(* Logix 5000 project; controller Receptivo vendor 1 type 14 code 106 rev 30.11; software revision 30.00; part 7 of 10 *)
(* tags used below, declared in another part *)
   Final_Print_1 : BOOL;
   Final_Print_2 : BOOL;
   Final_Print_3 : BOOL;
   Final_Print_4 : BOOL;
   ons_imprimiendo : BOOL;
   ons_nuevo_dia : BOOL;
   ons_print1 : BOOL;
   ons_print1_aux : BOOL;
   ons_print2 : BOOL;
   ons_print2_2 : BOOL;
   ons_print3 : BOOL;
   ons_print3_aux : BOOL;
   ons_print4 : BOOL;
   ons_print4_aux : BOOL;
   Print1_Ejecute : BOOL;
   Print1_OK : BOOL;
   Print2_Ejecute : BOOL;
   Print2_OK : BOOL;
   Print3_Ejecute : BOOL;
   Print3_OK : BOOL;
   Print4_Ejecute : BOOL;
   Print4_OK : BOOL;
   Printing_1 : BOOL;
   Printing_2 : BOOL;
   Printing_3 : BOOL;
   Printing_4 : BOOL;
   Salida_Cola_Est_1 : UDT_COLA;
   Salida_Cola_Est_2 : UDT_COLA;
   Salida_Cola_Est_3 : UDT_COLA;
   Salida_Cola_Est_4 : UDT_COLA;
   Actualiza1_Timer : TIMER;
   Actualiza2_Timer : TIMER;
   Actualiza3_Timer : TIMER;
   Actualiza4_Timer : TIMER;
   Actualiza_Reporte_1 : BOOL;
   Actualiza_Reporte_2 : BOOL;
   Actualiza_Reporte_3 : BOOL;
   Actualiza_Reporte_4 : BOOL;
   Ano_Biciesto : INT;
   Bit_Medianoche : BOOL;
   Cajas_Calculadas_Estacion_1 : REAL;
   Cajas_Calculadas_Estacion_2 : REAL;
   Cajas_Calculadas_Estacion_3 : REAL;
   Cajas_Calculadas_Estacion_4 : REAL;
   Cajas_CalculadasG_Estacion_1 : REAL;
   Cajas_CalculadasG_Estacion_2 : REAL;
   Cajas_CalculadasG_Estacion_3 : REAL;
   Cajas_CalculadasG_Estacion_4 : REAL;
   Calendario : Hora_y_Fecha;
   Cantidad_de_Productos : DINT;
   CINCO : SINT;
   Clima_1 : DINT;
   Cola_Estacion_1 : UDT_COLA[100];
   Cola_Estacion_1_A : UDT_COLA[100];
   Cola_Estacion_2 : UDT_COLA[100];
   Cola_Estacion_2_A : UDT_COLA[100];
   Cola_Estacion_3 : UDT_COLA[100];
   Cola_Estacion_3_A : UDT_COLA[100];
   Cola_Estacion_4 : UDT_COLA[100];
   Cola_Estacion_4_A : UDT_COLA[100];
   Consecutivo : INT;
   Contador_Consecutivo : COUNTER;
   Control_Cola_Est1 : CONTROL;
   Control_Cola_Est2 : CONTROL;
   Control_Cola_Est3 : CONTROL;
   Control_Cola_Est4 : CONTROL;
   Counter_R_Estacion1 : COUNTER;
   Counter_R_Estacion2 : COUNTER;
   Counter_R_Estacion3 : COUNTER;
   Counter_R_Estacion4 : COUNTER;
   CUATRO : SINT;
   Dia_del_Ano : INT;
   DOS : SINT;
   Espacios : STRING;
   Estacion_1_GCola : UDT_COLA;
   Estacion_1_GCola_1 : UDT_COLA;
   Estacion_1_General : UDT_GENERAL;
   Estacion_1_Resumen : UDT_COLA[20];
   Estacion_1_Resumen_A : UDT_COLA[20];
   Estacion_2_GCola : UDT_COLA;
   Estacion_2_GCola_1 : UDT_COLA;
   Estacion_2_General : UDT_GENERAL;
   Estacion_2_Resumen : UDT_COLA[20];
   Estacion_2_Resumen_A : UDT_COLA[20];
   Estacion_3_GCola : UDT_COLA;
   Estacion_3_GCola_1 : UDT_COLA;
   Estacion_3_General : UDT_GENERAL;
   Estacion_3_Resumen : UDT_COLA[20];
   Estacion_3_Resumen_A : UDT_COLA[20];
   Estacion_4_GCola : UDT_COLA;
   Estacion_4_GCola_1 : UDT_COLA;
   Estacion_4_General : UDT_GENERAL;
   Estacion_4_Resumen : UDT_COLA[20];
   Estacion_4_Resumen_A : UDT_COLA[20];
   Hoy : DINT;
   Impreso_1 : BOOL;
   Impreso_2 : BOOL;
   Impreso_3 : BOOL;
   Impreso_4 : BOOL;
   Imprimiendo_1 : BOOL;
   Imprimiendo_1_Timer : TIMER;
   Imprimiendo_2 : BOOL;
   Imprimiendo_2_Timer : TIMER;
   Imprimiendo_3 : BOOL;
   Imprimiendo_3_Timer : TIMER;
   Imprimiendo_4 : BOOL;
   Imprimiendo_4_Timer : TIMER;
   Index_Productos : DINT;
   Listado : INT;
   Listado_A : INT;
   Lote : DINT;
   Mes_dias : INT[13];
   new_day : BOOL;
   Num_Cajas_Reales_1 : DINT;
   Num_Cajas_Reales_2 : DINT;
   Num_Cajas_Reales_3 : DINT;
   Num_Cajas_Reales_4 : DINT;
   ons_add : BOOL;
   ons_add2 : BOOL;
   ons_add3 : BOOL;
   ons_add4 : BOOL;
   Ons_Corte_Dia : BOOL;
   Ons_NP : BOOL;
   Ons_NP2 : BOOL;
   Ons_NP3 : BOOL;
   Ons_NP4 : BOOL;
   ONS_Reporte_Dia : BOOL;
   Operador_1 : DINT;
   Peso_OK_Estacion_1 : BOOL;
   Peso_OK_Estacion_2 : BOOL;
   Peso_OK_Estacion_3 : BOOL;
   Peso_OK_Estacion_4 : BOOL;
   PESO_REAL_1 : DINT;
   PESO_REAL_2 : DINT;
   PESO_REAL_3 : DINT;
   PESO_REAL_4 : DINT;
   Print_1 : BOOL;
   Print_2 : BOOL;
   Print_3 : BOOL;
   Print_4 : BOOL;
   Printing_Enable : BOOL;
   Producto1 : UDT_Inventario;
   Producto2 : UDT_Inventario;
   Producto3 : UDT_Inventario;
   Producto4 : UDT_Inventario;
   Productos : UDT_Maestro[300];
   Prueba : UDT_COLA[3];
   Prueba_Bit : BOOL;
   Prueba_Index : DINT;
   Prueba_X : BOOL;
   QAD_Auxiliar_Est1 : STRING;
   QAD_Auxiliar_Est2 : STRING;
   QAD_Auxiliar_Est3 : STRING;
   QAD_Auxiliar_Est4 : STRING;
   Report_Con1 : BOOL;
   Reporte_Dia_Lach : BOOL;
   Reporte_Dia_Timer : TIMER;
   time_new : TIMER;
   TRES : SINT;
   try : BOOL;
   UNO : SINT;
   Zero : DINT;
(* MainProgram, continued *)

ROUTINE Impresion_1   (* ladder *)
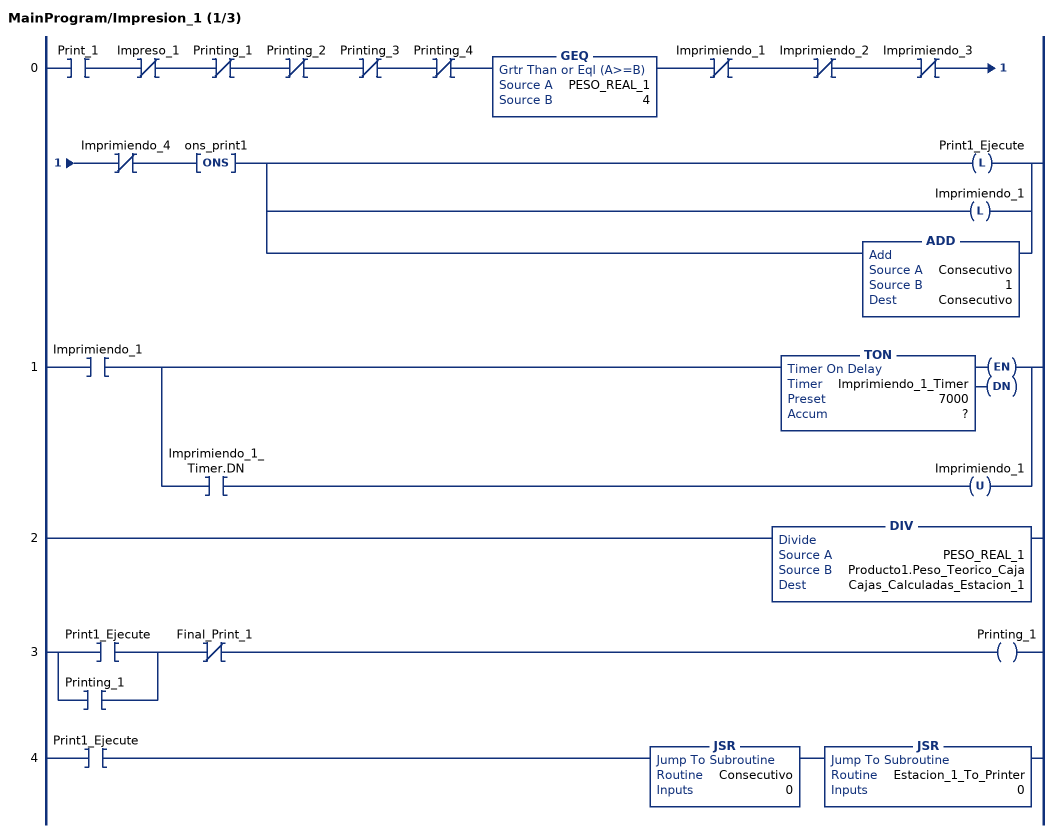
   0: XIC(Print_1)XIO(Impreso_1)XIO(Printing_1)XIO(Printing_2)XIO(Printing_3)XIO(Printing_4)GEQ(PESO_REAL_1,4)XIO(Imprimiendo_1)XIO(Imprimiendo_2)XIO(Imprimiendo_3)XIO(Imprimiendo_4)ONS(ons_print1)[OTL(Print1_Ejecute) ,OTL(Imprimiendo_1) ,ADD(Consecutivo,1,Consecutivo) ];
   1: XIC(Imprimiendo_1)[TON(Imprimiendo_1_Timer,?,?) ,XIC(Imprimiendo_1_Timer.DN) OTU(Imprimiendo_1) ];
   2: DIV(PESO_REAL_1,Producto1.Peso_Teorico_Caja,Cajas_Calculadas_Estacion_1);
   3: [XIC(Print1_Ejecute) ,XIC(Printing_1) ]XIO(Final_Print_1)OTE(Printing_1);
   4: XIC(Print1_Ejecute)JSR(Consecutivo,0)JSR(Estacion_1_To_Printer,0);
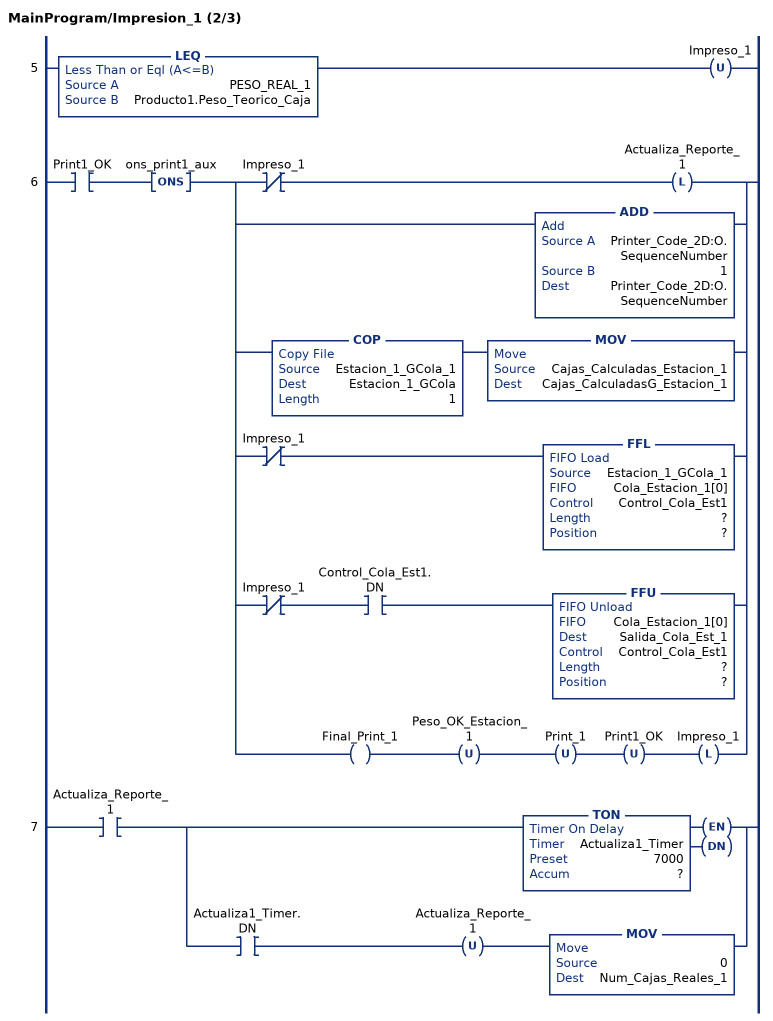
   5: LEQ(PESO_REAL_1,Producto1.Peso_Teorico_Caja)OTU(Impreso_1);
   6: XIC(Print1_OK)ONS(ons_print1_aux)[XIO(Impreso_1) OTL(Actualiza_Reporte_1) ,ADD(Printer_Code_2D:O.SequenceNumber,1,Printer_Code_2D:O.SequenceNumber) ,COP(Estacion_1_GCola_1,Estacion_1_GCola,1) MOV(Cajas_Calculadas_Estacion_1,Cajas_CalculadasG_Estacion_1) ,XIO(Impreso_1) FFL(Estacion_1_GCola_1,Cola_Estacion_1[0],Control_Cola_Est1,?,?) ,XIO(Impreso_1) XIC(Control_Cola_Est1.DN) FFU(Cola_Estacion_1[0],Salida_Cola_Est_1,Control_Cola_Est1,?,?) ,OTE(Final_Print_1) OTU(Peso_OK_Estacion_1) OTU(Print_1) OTU(Print1_OK) OTL(Impreso_1) ];
   7: XIC(Actualiza_Reporte_1)[TON(Actualiza1_Timer,?,?) ,XIC(Actualiza1_Timer.DN) OTU(Actualiza_Reporte_1) MOV(0,Num_Cajas_Reales_1) ];
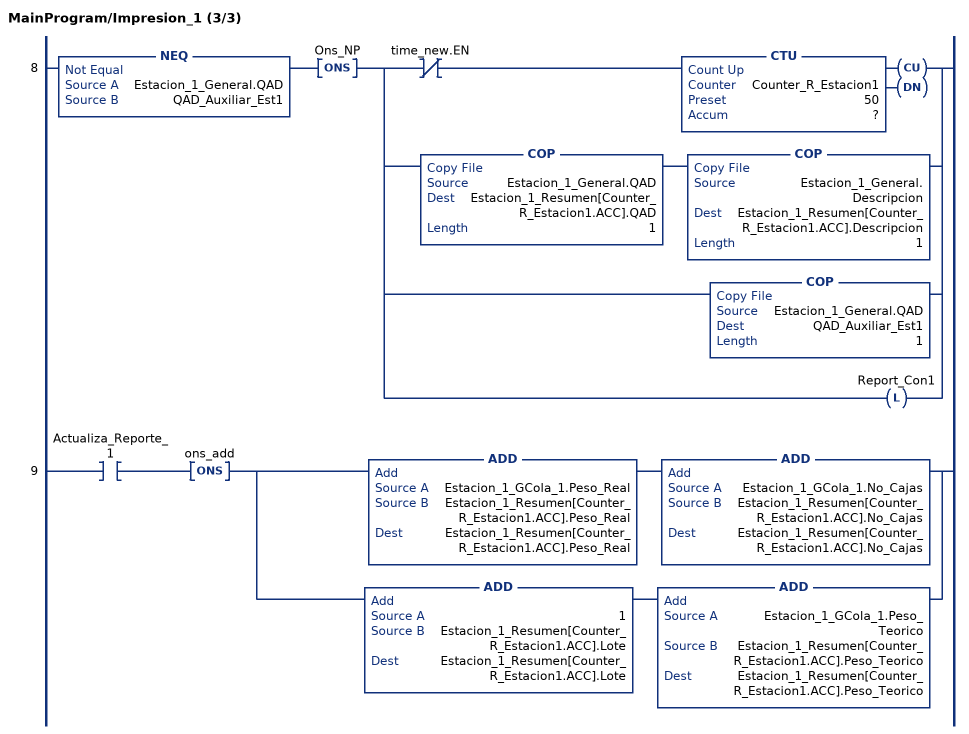
   8: NEQ(Estacion_1_General.QAD,QAD_Auxiliar_Est1)ONS(Ons_NP)[XIO(time_new.EN) CTU(Counter_R_Estacion1,?,?) ,COP(Estacion_1_General.QAD,Estacion_1_Resumen[Counter_R_Estacion1.ACC].QAD,1) COP(Estacion_1_General.Descripcion,Estacion_1_Resumen[Counter_R_Estacion1.ACC].Descripcion,1) ,COP(Estacion_1_General.QAD,QAD_Auxiliar_Est1,1) ,OTL(Report_Con1) ];
   9: XIC(Actualiza_Reporte_1)ONS(ons_add)[ADD(Estacion_1_GCola_1.Peso_Real,Estacion_1_Resumen[Counter_R_Estacion1.ACC].Peso_Real,Estacion_1_Resumen[Counter_R_Estacion1.ACC].Peso_Real) ADD(Estacion_1_GCola_1.No_Cajas,Estacion_1_Resumen[Counter_R_Estacion1.ACC].No_Cajas,Estacion_1_Resumen[Counter_R_Estacion1.ACC].No_Cajas) ,ADD(1,Estacion_1_Resumen[Counter_R_Estacion1.ACC].Lote,Estacion_1_Resumen[Counter_R_Estacion1.ACC].Lote) ADD(Estacion_1_GCola_1.Peso_Teorico,Estacion_1_Resumen[Counter_R_Estacion1.ACC].Peso_Teorico,Estacion_1_Resumen[Counter_R_Estacion1.ACC].Peso_Teorico) ];
END_ROUTINE

ROUTINE Impresion_2   (* ladder *)
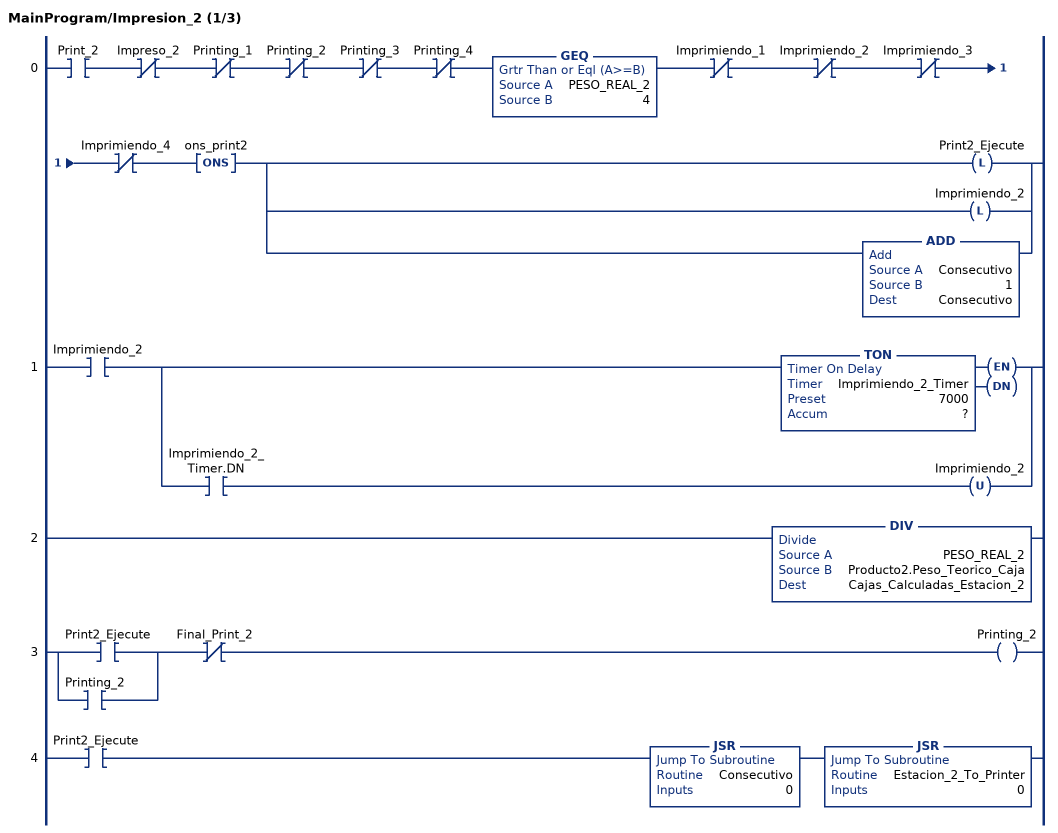
   0: XIC(Print_2)XIO(Impreso_2)XIO(Printing_1)XIO(Printing_2)XIO(Printing_3)XIO(Printing_4)GEQ(PESO_REAL_2,4)XIO(Imprimiendo_1)XIO(Imprimiendo_2)XIO(Imprimiendo_3)XIO(Imprimiendo_4)ONS(ons_print2)[OTL(Print2_Ejecute) ,OTL(Imprimiendo_2) ,ADD(Consecutivo,1,Consecutivo) ];
   1: XIC(Imprimiendo_2)[TON(Imprimiendo_2_Timer,?,?) ,XIC(Imprimiendo_2_Timer.DN) OTU(Imprimiendo_2) ];
   2: DIV(PESO_REAL_2,Producto2.Peso_Teorico_Caja,Cajas_Calculadas_Estacion_2);
   3: [XIC(Print2_Ejecute) ,XIC(Printing_2) ]XIO(Final_Print_2)OTE(Printing_2);
   4: XIC(Print2_Ejecute)JSR(Consecutivo,0)JSR(Estacion_2_To_Printer,0);
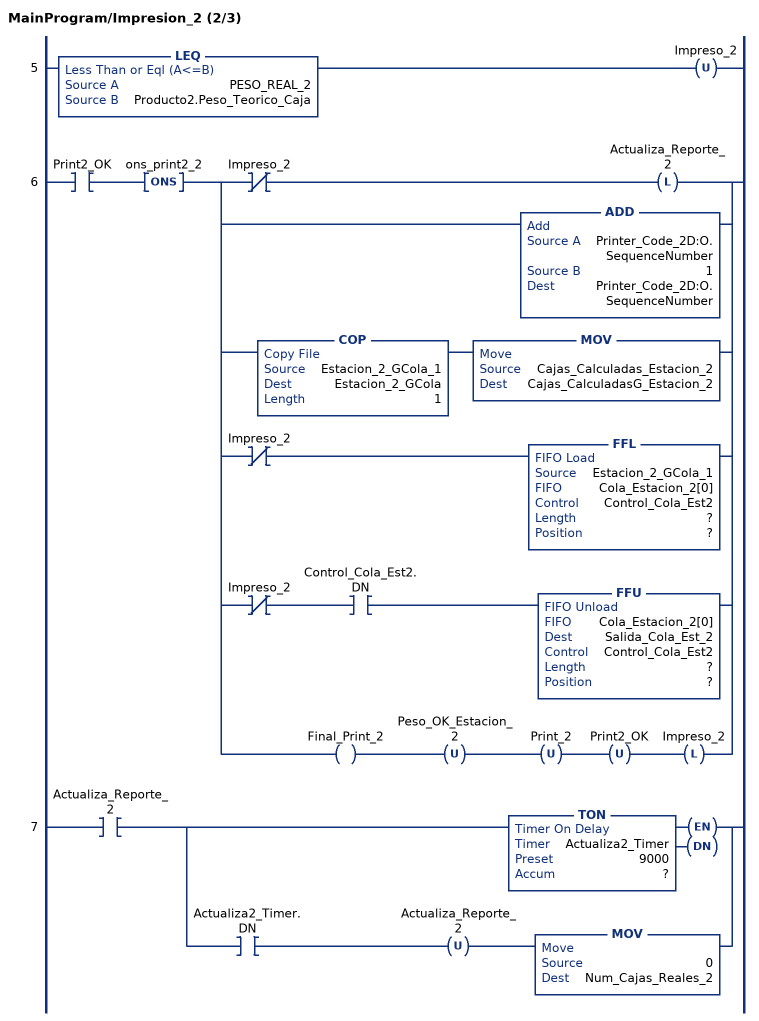
   5: LEQ(PESO_REAL_2,Producto2.Peso_Teorico_Caja)OTU(Impreso_2);
   6: XIC(Print2_OK)ONS(ons_print2_2)[XIO(Impreso_2) OTL(Actualiza_Reporte_2) ,ADD(Printer_Code_2D:O.SequenceNumber,1,Printer_Code_2D:O.SequenceNumber) ,COP(Estacion_2_GCola_1,Estacion_2_GCola,1) MOV(Cajas_Calculadas_Estacion_2,Cajas_CalculadasG_Estacion_2) ,XIO(Impreso_2) FFL(Estacion_2_GCola_1,Cola_Estacion_2[0],Control_Cola_Est2,?,?) ,XIO(Impreso_2) XIC(Control_Cola_Est2.DN) FFU(Cola_Estacion_2[0],Salida_Cola_Est_2,Control_Cola_Est2,?,?) ,OTE(Final_Print_2) OTU(Peso_OK_Estacion_2) OTU(Print_2) OTU(Print2_OK) OTL(Impreso_2) ];
   7: XIC(Actualiza_Reporte_2)[TON(Actualiza2_Timer,?,?) ,XIC(Actualiza2_Timer.DN) OTU(Actualiza_Reporte_2) MOV(0,Num_Cajas_Reales_2) ];
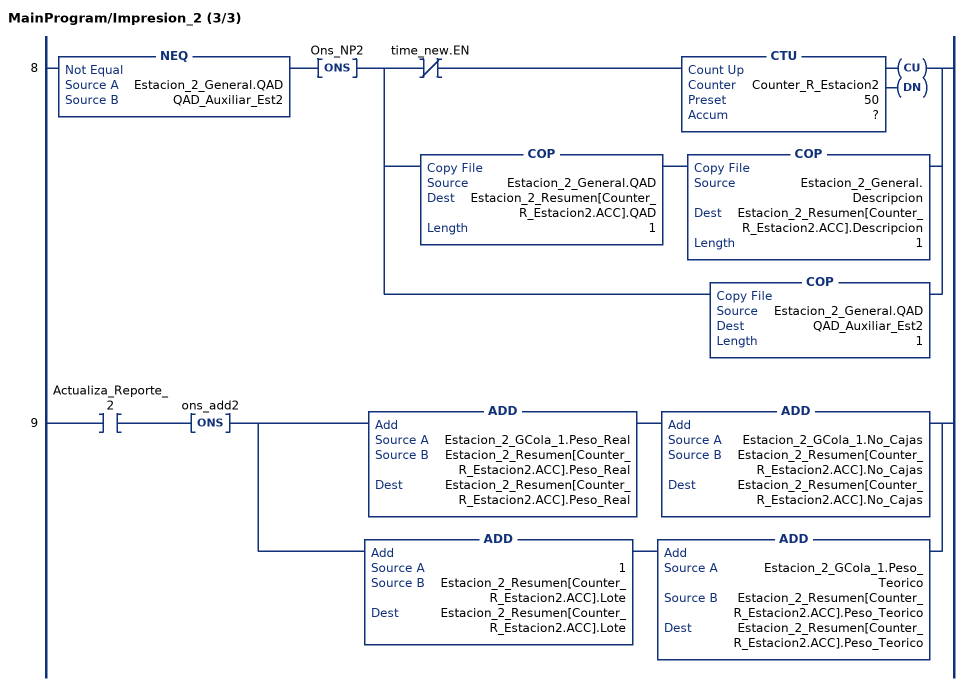
   8: NEQ(Estacion_2_General.QAD,QAD_Auxiliar_Est2)ONS(Ons_NP2)[XIO(time_new.EN) CTU(Counter_R_Estacion2,?,?) ,COP(Estacion_2_General.QAD,Estacion_2_Resumen[Counter_R_Estacion2.ACC].QAD,1) COP(Estacion_2_General.Descripcion,Estacion_2_Resumen[Counter_R_Estacion2.ACC].Descripcion,1) ,COP(Estacion_2_General.QAD,QAD_Auxiliar_Est2,1) ];
   9: XIC(Actualiza_Reporte_2)ONS(ons_add2)[ADD(Estacion_2_GCola_1.Peso_Real,Estacion_2_Resumen[Counter_R_Estacion2.ACC].Peso_Real,Estacion_2_Resumen[Counter_R_Estacion2.ACC].Peso_Real) ADD(Estacion_2_GCola_1.No_Cajas,Estacion_2_Resumen[Counter_R_Estacion2.ACC].No_Cajas,Estacion_2_Resumen[Counter_R_Estacion2.ACC].No_Cajas) ,ADD(1,Estacion_2_Resumen[Counter_R_Estacion2.ACC].Lote,Estacion_2_Resumen[Counter_R_Estacion2.ACC].Lote) ADD(Estacion_2_GCola_1.Peso_Teorico,Estacion_2_Resumen[Counter_R_Estacion2.ACC].Peso_Teorico,Estacion_2_Resumen[Counter_R_Estacion2.ACC].Peso_Teorico) ];
END_ROUTINE

ROUTINE Impresion_3   (* ladder *)
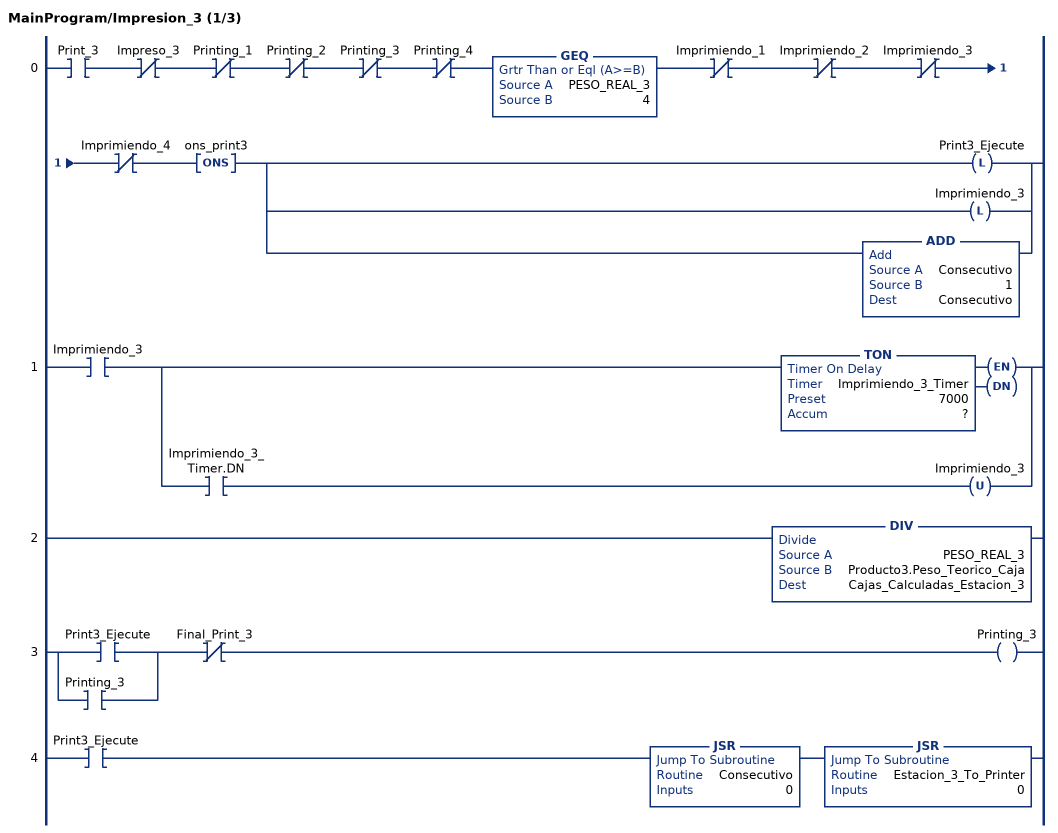
   0: XIC(Print_3)XIO(Impreso_3)XIO(Printing_1)XIO(Printing_2)XIO(Printing_3)XIO(Printing_4)GEQ(PESO_REAL_3,4)XIO(Imprimiendo_1)XIO(Imprimiendo_2)XIO(Imprimiendo_3)XIO(Imprimiendo_4)ONS(ons_print3)[OTL(Print3_Ejecute) ,OTL(Imprimiendo_3) ,ADD(Consecutivo,1,Consecutivo) ];
   1: XIC(Imprimiendo_3)[TON(Imprimiendo_3_Timer,?,?) ,XIC(Imprimiendo_3_Timer.DN) OTU(Imprimiendo_3) ];
   2: DIV(PESO_REAL_3,Producto3.Peso_Teorico_Caja,Cajas_Calculadas_Estacion_3);
   3: [XIC(Print3_Ejecute) ,XIC(Printing_3) ]XIO(Final_Print_3)OTE(Printing_3);
   4: XIC(Print3_Ejecute)JSR(Consecutivo,0)JSR(Estacion_3_To_Printer,0);
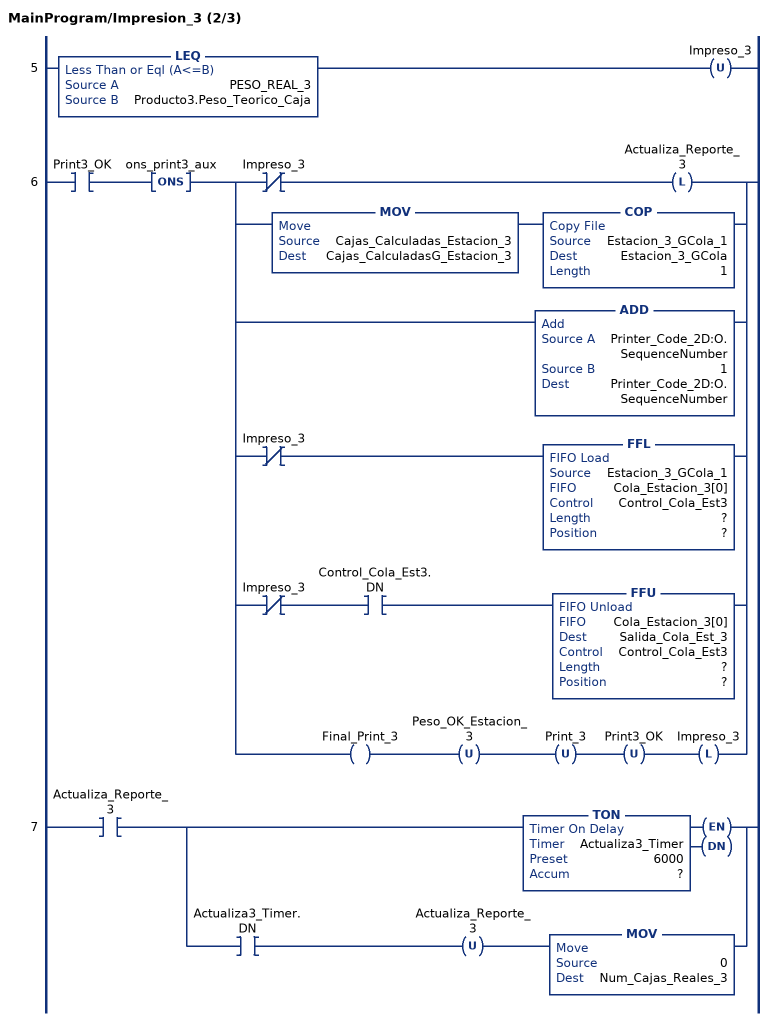
   5: LEQ(PESO_REAL_3,Producto3.Peso_Teorico_Caja)OTU(Impreso_3);
   6: XIC(Print3_OK)ONS(ons_print3_aux)[XIO(Impreso_3) OTL(Actualiza_Reporte_3) ,MOV(Cajas_Calculadas_Estacion_3,Cajas_CalculadasG_Estacion_3) COP(Estacion_3_GCola_1,Estacion_3_GCola,1) ,ADD(Printer_Code_2D:O.SequenceNumber,1,Printer_Code_2D:O.SequenceNumber) ,XIO(Impreso_3) FFL(Estacion_3_GCola_1,Cola_Estacion_3[0],Control_Cola_Est3,?,?) ,XIO(Impreso_3) XIC(Control_Cola_Est3.DN) FFU(Cola_Estacion_3[0],Salida_Cola_Est_3,Control_Cola_Est3,?,?) ,OTE(Final_Print_3) OTU(Peso_OK_Estacion_3) OTU(Print_3) OTU(Print3_OK) OTL(Impreso_3) ];
   7: XIC(Actualiza_Reporte_3)[TON(Actualiza3_Timer,?,?) ,XIC(Actualiza3_Timer.DN) OTU(Actualiza_Reporte_3) MOV(0,Num_Cajas_Reales_3) ];
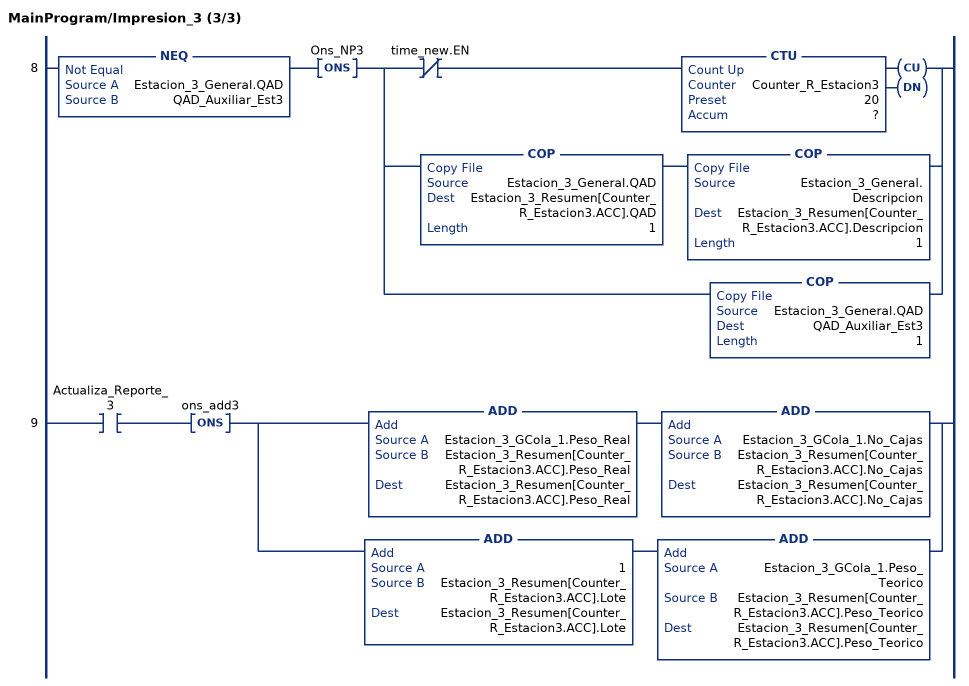
   8: NEQ(Estacion_3_General.QAD,QAD_Auxiliar_Est3)ONS(Ons_NP3)[XIO(time_new.EN) CTU(Counter_R_Estacion3,?,?) ,COP(Estacion_3_General.QAD,Estacion_3_Resumen[Counter_R_Estacion3.ACC].QAD,1) COP(Estacion_3_General.Descripcion,Estacion_3_Resumen[Counter_R_Estacion3.ACC].Descripcion,1) ,COP(Estacion_3_General.QAD,QAD_Auxiliar_Est3,1) ];
   9: XIC(Actualiza_Reporte_3)ONS(ons_add3)[ADD(Estacion_3_GCola_1.Peso_Real,Estacion_3_Resumen[Counter_R_Estacion3.ACC].Peso_Real,Estacion_3_Resumen[Counter_R_Estacion3.ACC].Peso_Real) ADD(Estacion_3_GCola_1.No_Cajas,Estacion_3_Resumen[Counter_R_Estacion3.ACC].No_Cajas,Estacion_3_Resumen[Counter_R_Estacion3.ACC].No_Cajas) ,ADD(1,Estacion_3_Resumen[Counter_R_Estacion3.ACC].Lote,Estacion_3_Resumen[Counter_R_Estacion3.ACC].Lote) ADD(Estacion_3_GCola_1.Peso_Teorico,Estacion_3_Resumen[Counter_R_Estacion3.ACC].Peso_Teorico,Estacion_3_Resumen[Counter_R_Estacion3.ACC].Peso_Teorico) ];
END_ROUTINE

ROUTINE Impresion_4   (* ladder *)
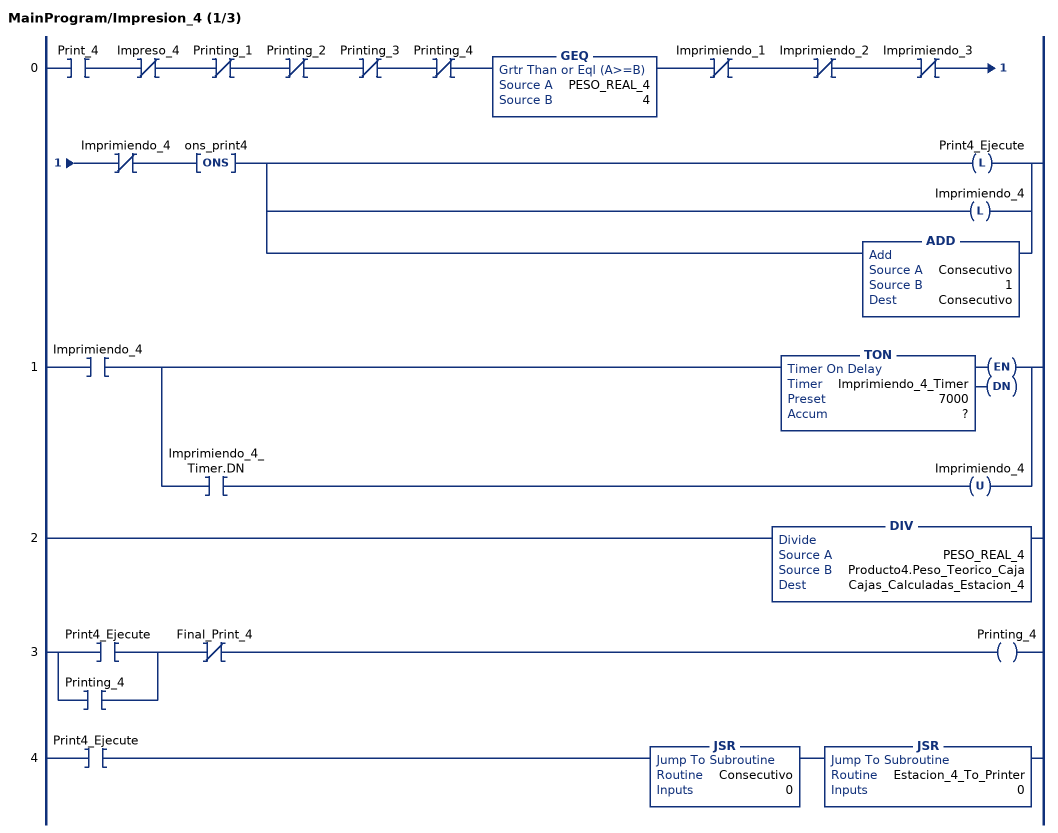
   0: XIC(Print_4)XIO(Impreso_4)XIO(Printing_1)XIO(Printing_2)XIO(Printing_3)XIO(Printing_4)GEQ(PESO_REAL_4,4)XIO(Imprimiendo_1)XIO(Imprimiendo_2)XIO(Imprimiendo_3)XIO(Imprimiendo_4)ONS(ons_print4)[OTL(Print4_Ejecute) ,OTL(Imprimiendo_4) ,ADD(Consecutivo,1,Consecutivo) ];
   1: XIC(Imprimiendo_4)[TON(Imprimiendo_4_Timer,?,?) ,XIC(Imprimiendo_4_Timer.DN) OTU(Imprimiendo_4) ];
   2: DIV(PESO_REAL_4,Producto4.Peso_Teorico_Caja,Cajas_Calculadas_Estacion_4);
   3: [XIC(Print4_Ejecute) ,XIC(Printing_4) ]XIO(Final_Print_4)OTE(Printing_4);
   4: XIC(Print4_Ejecute)JSR(Consecutivo,0)JSR(Estacion_4_To_Printer,0);
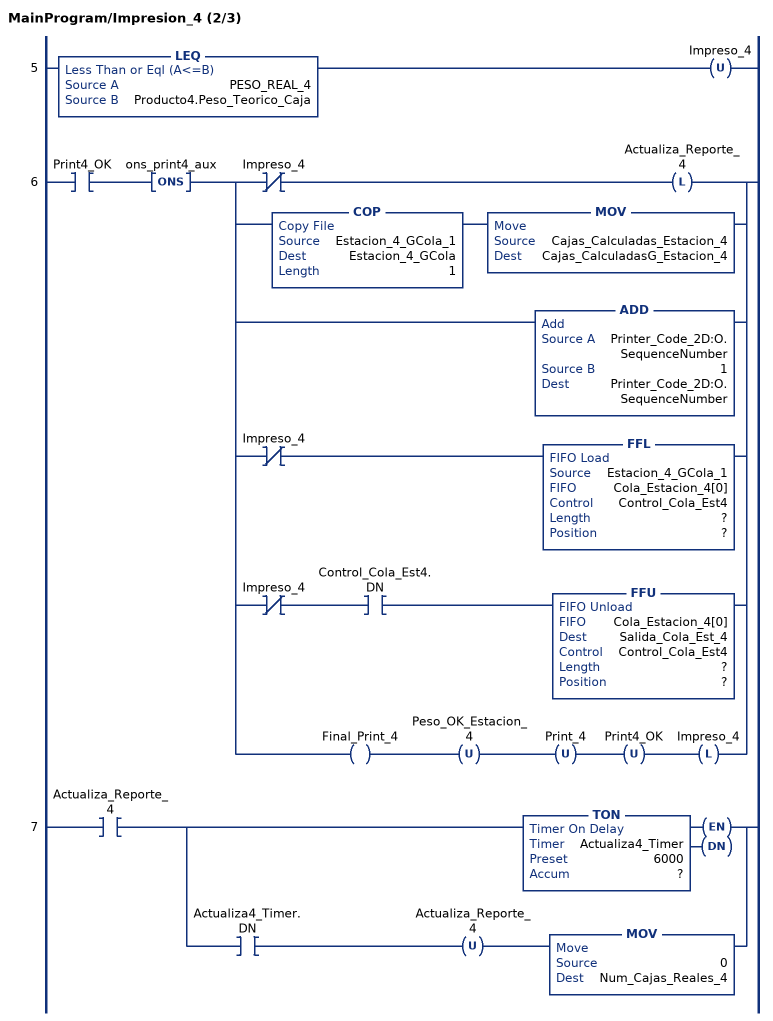
   5: LEQ(PESO_REAL_4,Producto4.Peso_Teorico_Caja)OTU(Impreso_4);
   6: XIC(Print4_OK)ONS(ons_print4_aux)[XIO(Impreso_4) OTL(Actualiza_Reporte_4) ,COP(Estacion_4_GCola_1,Estacion_4_GCola,1) MOV(Cajas_Calculadas_Estacion_4,Cajas_CalculadasG_Estacion_4) ,ADD(Printer_Code_2D:O.SequenceNumber,1,Printer_Code_2D:O.SequenceNumber) ,XIO(Impreso_4) FFL(Estacion_4_GCola_1,Cola_Estacion_4[0],Control_Cola_Est4,?,?) ,XIO(Impreso_4) XIC(Control_Cola_Est4.DN) FFU(Cola_Estacion_4[0],Salida_Cola_Est_4,Control_Cola_Est4,?,?) ,OTE(Final_Print_4) OTU(Peso_OK_Estacion_4) OTU(Print_4) OTU(Print4_OK) OTL(Impreso_4) ];
   7: XIC(Actualiza_Reporte_4)[TON(Actualiza4_Timer,?,?) ,XIC(Actualiza4_Timer.DN) OTU(Actualiza_Reporte_4) MOV(0,Num_Cajas_Reales_4) ];
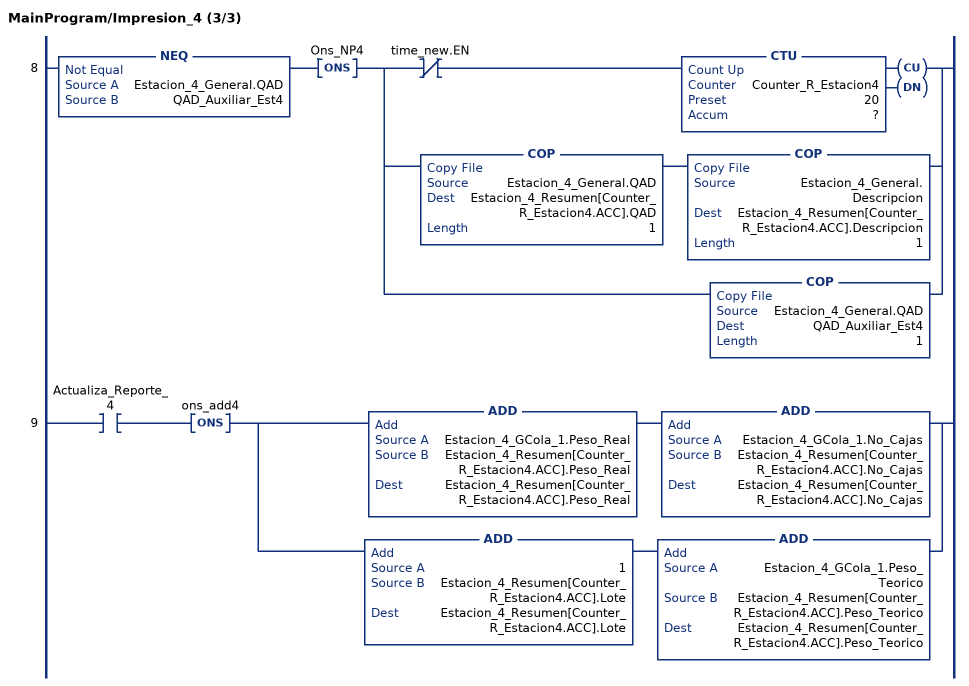
   8: NEQ(Estacion_4_General.QAD,QAD_Auxiliar_Est4)ONS(Ons_NP4)[XIO(time_new.EN) CTU(Counter_R_Estacion4,?,?) ,COP(Estacion_4_General.QAD,Estacion_4_Resumen[Counter_R_Estacion4.ACC].QAD,1) COP(Estacion_4_General.Descripcion,Estacion_4_Resumen[Counter_R_Estacion4.ACC].Descripcion,1) ,COP(Estacion_4_General.QAD,QAD_Auxiliar_Est4,1) ];
   9: XIC(Actualiza_Reporte_4)ONS(ons_add4)[ADD(Estacion_4_GCola_1.Peso_Real,Estacion_4_Resumen[Counter_R_Estacion4.ACC].Peso_Real,Estacion_4_Resumen[Counter_R_Estacion4.ACC].Peso_Real) ADD(Estacion_4_GCola_1.No_Cajas,Estacion_4_Resumen[Counter_R_Estacion4.ACC].No_Cajas,Estacion_4_Resumen[Counter_R_Estacion4.ACC].No_Cajas) ,ADD(1,Estacion_4_Resumen[Counter_R_Estacion4.ACC].Lote,Estacion_4_Resumen[Counter_R_Estacion4.ACC].Lote) ADD(Estacion_4_GCola_1.Peso_Teorico,Estacion_4_Resumen[Counter_R_Estacion4.ACC].Peso_Teorico,Estacion_4_Resumen[Counter_R_Estacion4.ACC].Peso_Teorico) ];
END_ROUTINE

ROUTINE MainRoutine   (* ladder *)
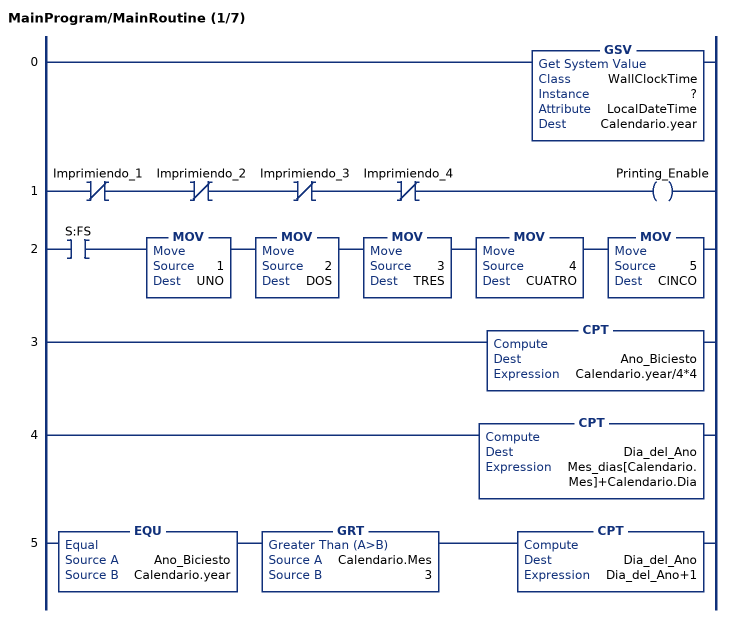
   0: GSV(WallClockTime,?,LocalDateTime,Calendario.year);
   1: XIO(Imprimiendo_1)XIO(Imprimiendo_2)XIO(Imprimiendo_3)XIO(Imprimiendo_4)OTE(Printing_Enable);
   2: XIC(S:FS)MOV(1,UNO)MOV(2,DOS)MOV(3,TRES)MOV(4,CUATRO)MOV(5,CINCO);
   3: CPT(Ano_Biciesto,Calendario.year/4*4);
   4: CPT(Dia_del_Ano,Mes_dias[Calendario.Mes]+Calendario.Dia);
   5: EQU(Ano_Biciesto,Calendario.year)GRT(Calendario.Mes,3)CPT(Dia_del_Ano,Dia_del_Ano+1);
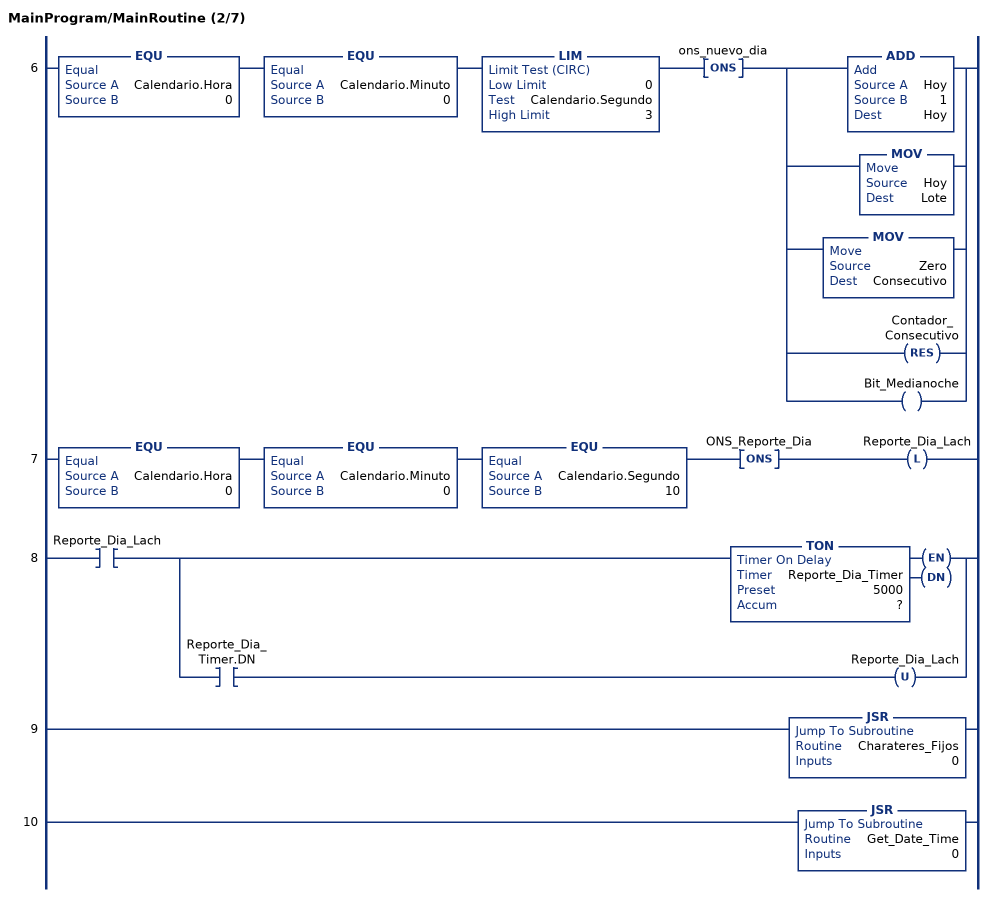
   6: EQU(Calendario.Hora,0)EQU(Calendario.Minuto,0)LIM(0,Calendario.Segundo,3)ONS(ons_nuevo_dia)[ADD(Hoy,1,Hoy) ,MOV(Hoy,Lote) ,MOV(Zero,Consecutivo) ,RES(Contador_Consecutivo) ,OTE(Bit_Medianoche) ];
   7: EQU(Calendario.Hora,0)EQU(Calendario.Minuto,0)EQU(Calendario.Segundo,10)ONS(ONS_Reporte_Dia)OTL(Reporte_Dia_Lach);
   8: XIC(Reporte_Dia_Lach)[TON(Reporte_Dia_Timer,?,?) ,XIC(Reporte_Dia_Timer.DN) OTU(Reporte_Dia_Lach) ];
   9: JSR(Charateres_Fijos,0);
   10: JSR(Get_Date_Time,0);
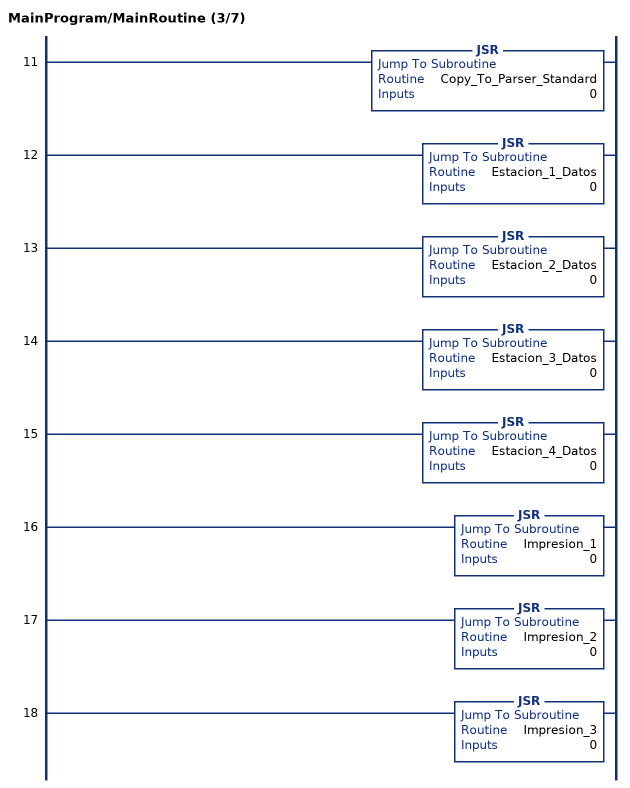
   11: JSR(Copy_To_Parser_Standard,0);
   12: JSR(Estacion_1_Datos,0);
   13: JSR(Estacion_2_Datos,0);
   14: JSR(Estacion_3_Datos,0);
   15: JSR(Estacion_4_Datos,0);
   16: JSR(Impresion_1,0);
   17: JSR(Impresion_2,0);
   18: JSR(Impresion_3,0);
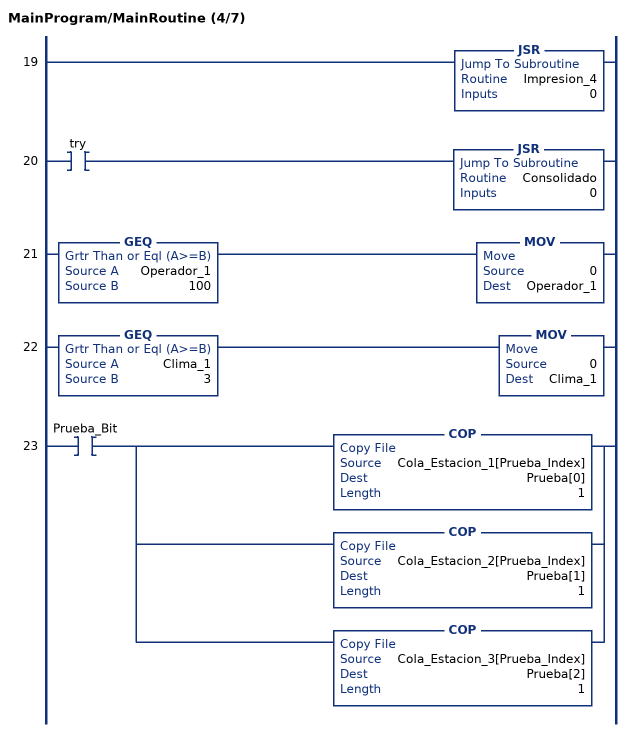
   19: JSR(Impresion_4,0);
   20: XIC(try)JSR(Consolidado,0);
   21: GEQ(Operador_1,100)MOV(0,Operador_1);
   22: GEQ(Clima_1,3)MOV(0,Clima_1);
   23: XIC(Prueba_Bit)[COP(Cola_Estacion_1[Prueba_Index],Prueba[0],1) ,COP(Cola_Estacion_2[Prueba_Index],Prueba[1],1) ,COP(Cola_Estacion_3[Prueba_Index],Prueba[2],1) ];
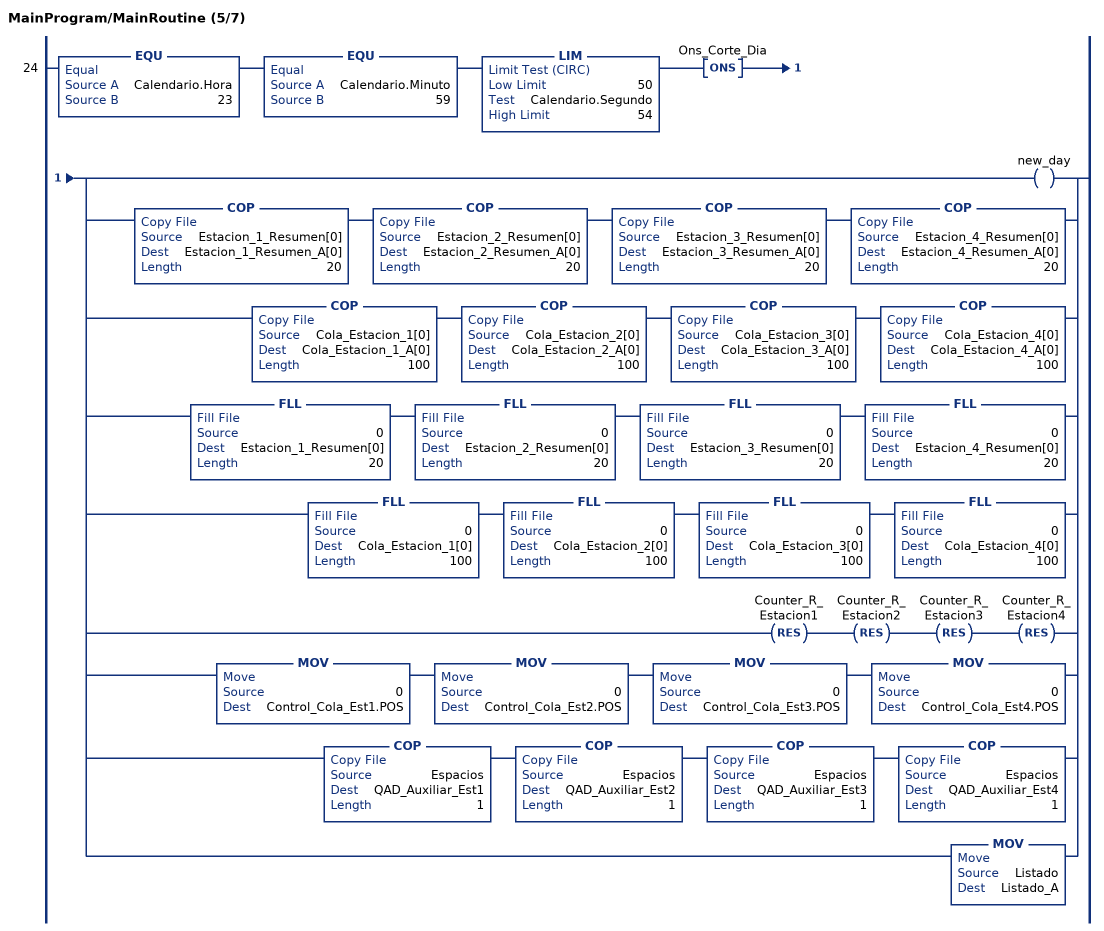
   24: EQU(Calendario.Hora,23)EQU(Calendario.Minuto,59)LIM(50,Calendario.Segundo,54)ONS(Ons_Corte_Dia)[OTE(new_day) ,COP(Estacion_1_Resumen[0],Estacion_1_Resumen_A[0],20) COP(Estacion_2_Resumen[0],Estacion_2_Resumen_A[0],20) COP(Estacion_3_Resumen[0],Estacion_3_Resumen_A[0],20) COP(Estacion_4_Resumen[0],Estacion_4_Resumen_A[0],20) ,COP(Cola_Estacion_1[0],Cola_Estacion_1_A[0],100) COP(Cola_Estacion_2[0],Cola_Estacion_2_A[0],100) COP(Cola_Estacion_3[0],Cola_Estacion_3_A[0],100) COP(Cola_Estacion_4[0],Cola_Estacion_4_A[0],100) ,FLL(0,Estacion_1_Resumen[0],20) FLL(0,Estacion_2_Resumen[0],20) FLL(0,Estacion_3_Resumen[0],20) FLL(0,Estacion_4_Resumen[0],20) ,FLL(0,Cola_Estacion_1[0],100) FLL(0,Cola_Estacion_2[0],100) FLL(0,Cola_Estacion_3[0],100) FLL(0,Cola_Estacion_4[0],100) ,RES(Counter_R_Estacion1) RES(Counter_R_Estacion2) RES(Counter_R_Estacion3) RES(Counter_R_Estacion4) ,MOV(0,Control_Cola_Est1.POS) MOV(0,Control_Cola_Est2.POS) MOV(0,Control_Cola_Est3.POS) MOV(0,Control_Cola_Est4.POS) ,COP(Espacios,QAD_Auxiliar_Est1,1) COP(Espacios,QAD_Auxiliar_Est2,1) COP(Espacios,QAD_Auxiliar_Est3,1) COP(Espacios,QAD_Auxiliar_Est4,1) ,MOV(Listado,Listado_A) ];
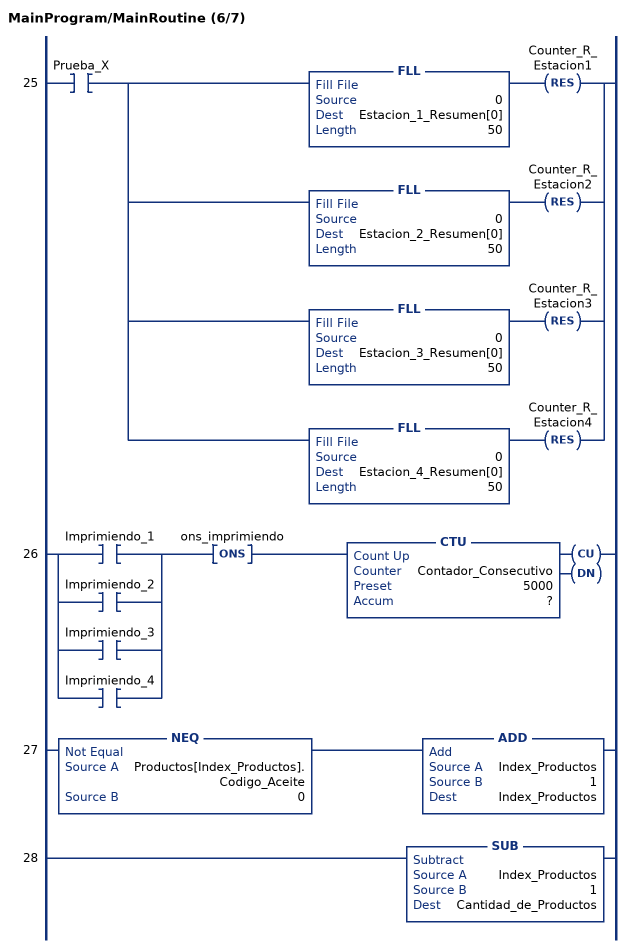
   25: XIC(Prueba_X)[FLL(0,Estacion_1_Resumen[0],50) RES(Counter_R_Estacion1) ,FLL(0,Estacion_2_Resumen[0],50) RES(Counter_R_Estacion2) ,FLL(0,Estacion_3_Resumen[0],50) RES(Counter_R_Estacion3) ,FLL(0,Estacion_4_Resumen[0],50) RES(Counter_R_Estacion4) ];
   26: [XIC(Imprimiendo_1) ,XIC(Imprimiendo_2) ,XIC(Imprimiendo_3) ,XIC(Imprimiendo_4) ]ONS(ons_imprimiendo)CTU(Contador_Consecutivo,?,?);
   27: NEQ(Productos[Index_Productos].Codigo_Aceite,0)ADD(Index_Productos,1,Index_Productos);
   28: SUB(Index_Productos,1,Cantidad_de_Productos);
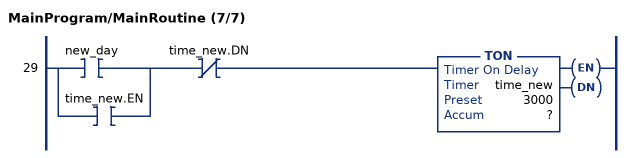
   29: [XIC(new_day) ,XIC(time_new.EN) ]XIO(time_new.DN)TON(time_new,?,?);
END_ROUTINE
END_PROGRAM
